PROGRAM MAIN
VAR
END_VAR

ReadAnalogInput();

END_PROGRAM

(* stored: Version 1.1.0.1, ProductVersion 3.1.4024.12
   POU MAIN: Id {51e18e0a-bf97-43bb-bd25-74158815971f}, SpecialFunc None *)
